// TIA Portal V19 export
TYPE "XYZ_Coordinates"
   STRUCT
      X : Int;
      Y : Int;
      Z : Int;
      Mode : Int;
   END_STRUCT;
END_TYPE
